Yaskawa INFORM job: ABRE_GRAMPOS.JBI

/JOB
//NAME ABRE_GRAMPOS
///FOLDERNAME GRAMPOS
//POS
///NPOS 0,0,0,0,0,0
//INST
///DATE 2022/06/09 09:24
///ATTR SC,RW
NOP
DOUT OT#(537) OFF
DOUT OT#(538) ON
WAIT IN#(537)=ON
WAIT IN#(539)=ON
WAIT IN#(541)=ON
WAIT IN#(543)=ON
END
